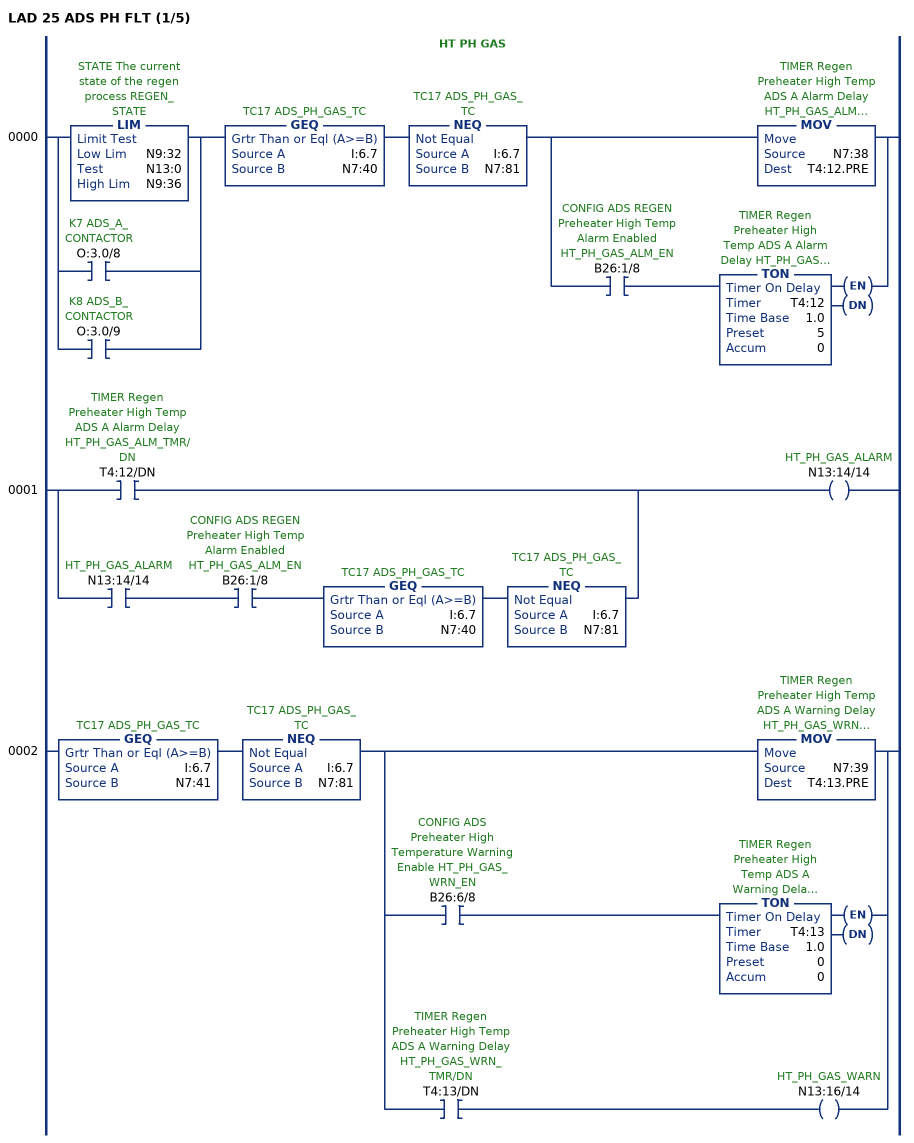
% Rung: 0 %
% TITLE: HT PH GAS %
SOR BST LIM N9:32 N13:0 N9:36 NXB XIC O:3.0/8 NXB XIC O:3.0/9 BND GEQ I:6.7 N7:40 NEQ I:6.7 N7:81 BST MOV N7:38 T4:12.PRE NXB XIC B26:1/8 TON T4:12 1.0 5 0 BND EOR
%   N9:32  REGEN_VENT  "STATE Regen Vent" %
%   N13:0  REGEN_STATE  "STATE The current state of the regen process" %
%   N9:36  REGEN_COOL  "STATE Regen Cool" %
%   O:3.0/8  ADS_A_CONTACTOR  "K7" %
%   O:3.0/9  ADS_B_CONTACTOR  "K8" %
%   I:6.7  ADS_PH_GAS_TC  "TC17" %
%   N7:40  HT_PH_GAS_ALM_SP  "CONFIG ADS Preheater High Temperature Alarm Temperature" %
%   N7:81  TC_OPEN_SP  "CONFIG The value read by an open TC input" %
%   N7:38  HT_PH_GAS_ALM_DLY  "CONFIG ADS Preheater High Temperature Alarm Delay" %
%   T4:12  HT_PH_GAS_ALM_TMR  "TIMER Regen Preheater High Temp ADS A Alarm Delay" %
%   B26:1/8  HT_PH_GAS_ALM_EN  "CONFIG ADS REGEN Preheater High Temp Alarm Enabled" %
% Rung: 1 %
SOR BST XIC T4:12/DN NXB XIC N13:14/14 XIC B26:1/8 GEQ I:6.7 N7:40 NEQ I:6.7 N7:81 BND OTE N13:14/14 EOR
%   T4:12  HT_PH_GAS_ALM_TMR  "TIMER Regen Preheater High Temp ADS A Alarm Delay" %
%   N13:14/14  HT_PH_GAS_ALARM %
%   B26:1/8  HT_PH_GAS_ALM_EN  "CONFIG ADS REGEN Preheater High Temp Alarm Enabled" %
%   I:6.7  ADS_PH_GAS_TC  "TC17" %
%   N7:40  HT_PH_GAS_ALM_SP  "CONFIG ADS Preheater High Temperature Alarm Temperature" %
%   N7:81  TC_OPEN_SP  "CONFIG The value read by an open TC input" %
% Rung: 2 %
SOR GEQ I:6.7 N7:41 NEQ I:6.7 N7:81 BST MOV N7:39 T4:13.PRE NXB XIC B26:6/8 TON T4:13 1.0 0 0 NXB XIC T4:13/DN OTE N13:16/14 BND EOR
%   I:6.7  ADS_PH_GAS_TC  "TC17" %
%   N7:41  HT_PH_GAS_WRN_SP  "CONFIG ADS Preheater High Temperature Warning Temperature" %
%   N7:81  TC_OPEN_SP  "CONFIG The value read by an open TC input" %
%   N7:39  HT_PH_GAS_WRN_DLY  "CONFIG ADS Preheater High Temperature Warning Delay" %
%   T4:13  HT_PH_GAS_WRN_TMR  "TIMER Regen Preheater High Temp ADS A Warning Delay" %
%   B26:6/8  HT_PH_GAS_WRN_EN  "CONFIG ADS Preheater High Temperature Warning Enable" %
%   N13:16/14  HT_PH_GAS_WARN %

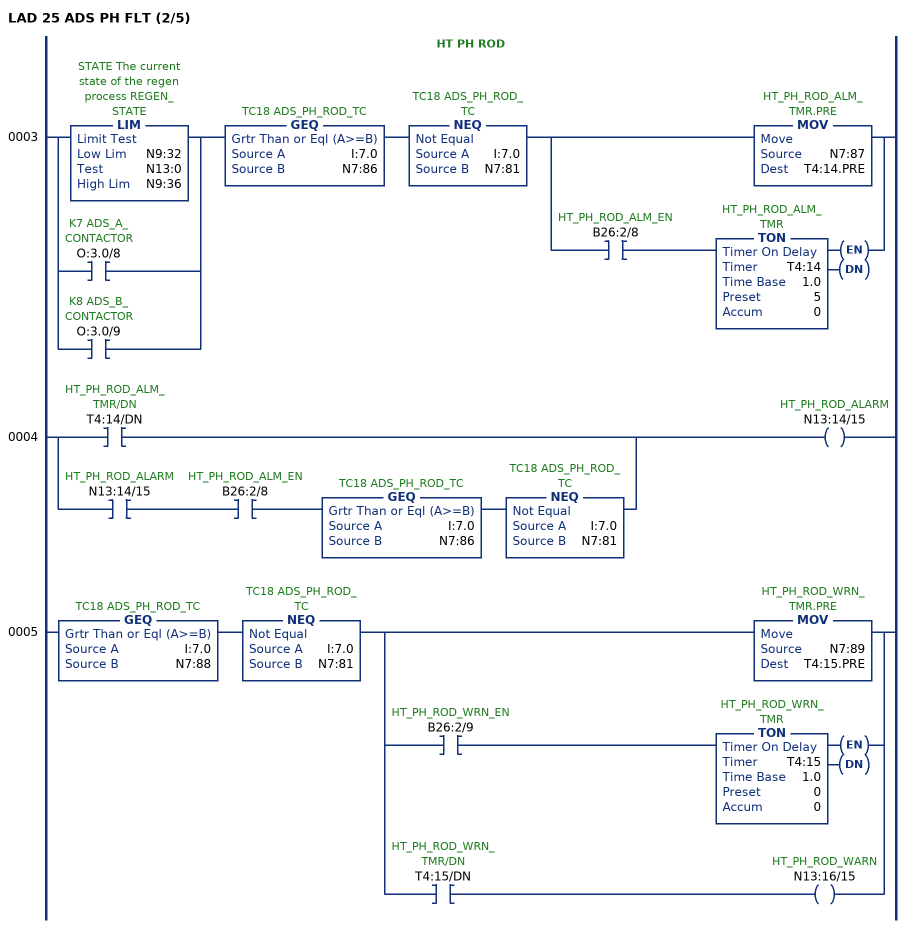
% Rung: 3 %
% TITLE: HT PH ROD %
SOR BST LIM N9:32 N13:0 N9:36 NXB XIC O:3.0/8 NXB XIC O:3.0/9 BND GEQ I:7.0 N7:86 NEQ I:7.0 N7:81 BST MOV N7:87 T4:14.PRE NXB XIC B26:2/8 TON T4:14 1.0 5 0 BND EOR
%   N9:32  REGEN_VENT  "STATE Regen Vent" %
%   N13:0  REGEN_STATE  "STATE The current state of the regen process" %
%   N9:36  REGEN_COOL  "STATE Regen Cool" %
%   O:3.0/8  ADS_A_CONTACTOR  "K7" %
%   O:3.0/9  ADS_B_CONTACTOR  "K8" %
%   I:7.0  ADS_PH_ROD_TC  "TC18" %
%   N7:86  HT_PH_ROD_ALM_SP %
%   N7:81  TC_OPEN_SP  "CONFIG The value read by an open TC input" %
%   N7:87  HT_PH_ROD_ALM_DLY %
%   T4:14  HT_PH_ROD_ALM_TMR %
%   B26:2/8  HT_PH_ROD_ALM_EN %
% Rung: 4 %
SOR BST XIC T4:14/DN NXB XIC N13:14/15 XIC B26:2/8 GEQ I:7.0 N7:86 NEQ I:7.0 N7:81 BND OTE N13:14/15 EOR
%   T4:14  HT_PH_ROD_ALM_TMR %
%   N13:14/15  HT_PH_ROD_ALARM %
%   B26:2/8  HT_PH_ROD_ALM_EN %
%   I:7.0  ADS_PH_ROD_TC  "TC18" %
%   N7:86  HT_PH_ROD_ALM_SP %
%   N7:81  TC_OPEN_SP  "CONFIG The value read by an open TC input" %
% Rung: 5 %
SOR GEQ I:7.0 N7:88 NEQ I:7.0 N7:81 BST MOV N7:89 T4:15.PRE NXB XIC B26:2/9 TON T4:15 1.0 0 0 NXB XIC T4:15/DN OTE N13:16/15 BND EOR
%   I:7.0  ADS_PH_ROD_TC  "TC18" %
%   N7:88  HT_PH_ROD_WRN_SP %
%   N7:81  TC_OPEN_SP  "CONFIG The value read by an open TC input" %
%   N7:89  HT_PH_ROD_WRN_DLY %
%   T4:15  HT_PH_ROD_WRN_TMR %
%   B26:2/9  HT_PH_ROD_WRN_EN %
%   N13:16/15  HT_PH_ROD_WARN %

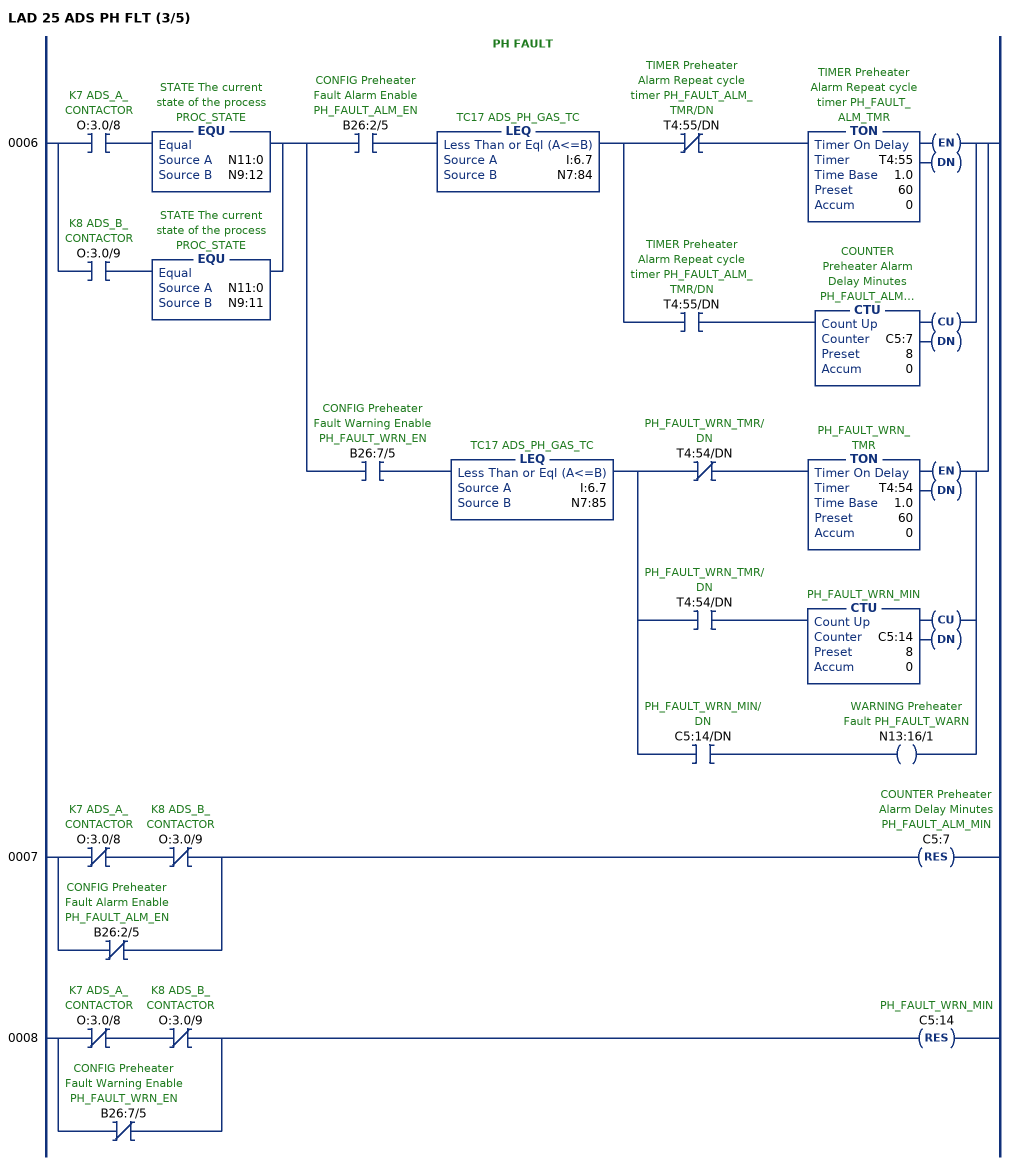
% Rung: 6 %
% TITLE: PH FAULT %
SOR BST XIC O:3.0/8 EQU N11:0 N9:12 NXB XIC O:3.0/9 EQU N11:0 N9:11 BND BST XIC B26:2/5 LEQ I:6.7 N7:84 BST XIO T4:55/DN TON T4:55 1.0 60 0 NXB XIC T4:55/DN CTU C5:7 8 0 BND NXB XIC B26:7/5 LEQ I:6.7 N7:85 BST XIO T4:54/DN TON T4:54 1.0 60 0 NXB XIC T4:54/DN CTU C5:14 8 0 NXB XIC C5:14/DN OTE N13:16/1 BND BND EOR
%   O:3.0/8  ADS_A_CONTACTOR  "K7" %
%   N11:0  PROC_STATE  "STATE The current state of the process" %
%   N9:12  PROC_PFY_B_REG_A  "STATE Process Purify B" %
%   O:3.0/9  ADS_B_CONTACTOR  "K8" %
%   N9:11  PROC_PFY_A_REG_B  "STATE Process Purify A" %
%   B26:2/5  PH_FAULT_ALM_EN  "CONFIG Preheater Fault Alarm Enable" %
%   I:6.7  ADS_PH_GAS_TC  "TC17" %
%   N7:84  PH_FAULT_ALARM_SP  "CONFIG Preheater Temperature Delta Alarm Setpoint" %
%   T4:55  PH_FAULT_ALM_TMR  "TIMER Preheater Alarm Repeat cycle timer" %
%   C5:7  PH_FAULT_ALM_MIN  "COUNTER Preheater Alarm Delay Minutes" %
%   B26:7/5  PH_FAULT_WRN_EN  "CONFIG Preheater Fault Warning Enable" %
%   N7:85  PH_FAULT_WARN_SP %
%   T4:54  PH_FAULT_WRN_TMR %
%   C5:14  PH_FAULT_WRN_MIN %
%   N13:16/1  PH_FAULT_WARN  "WARNING Preheater Fault" %
% Rung: 7 %
SOR BST XIO O:3.0/8 XIO O:3.0/9 NXB XIO B26:2/5 BND RES C5:7 EOR
%   O:3.0/8  ADS_A_CONTACTOR  "K7" %
%   O:3.0/9  ADS_B_CONTACTOR  "K8" %
%   B26:2/5  PH_FAULT_ALM_EN  "CONFIG Preheater Fault Alarm Enable" %
%   C5:7  PH_FAULT_ALM_MIN  "COUNTER Preheater Alarm Delay Minutes" %
% Rung: 8 %
SOR BST XIO O:3.0/8 XIO O:3.0/9 NXB XIO B26:7/5 BND RES C5:14 EOR
%   O:3.0/8  ADS_A_CONTACTOR  "K7" %
%   O:3.0/9  ADS_B_CONTACTOR  "K8" %
%   B26:7/5  PH_FAULT_WRN_EN  "CONFIG Preheater Fault Warning Enable" %
%   C5:14  PH_FAULT_WRN_MIN %

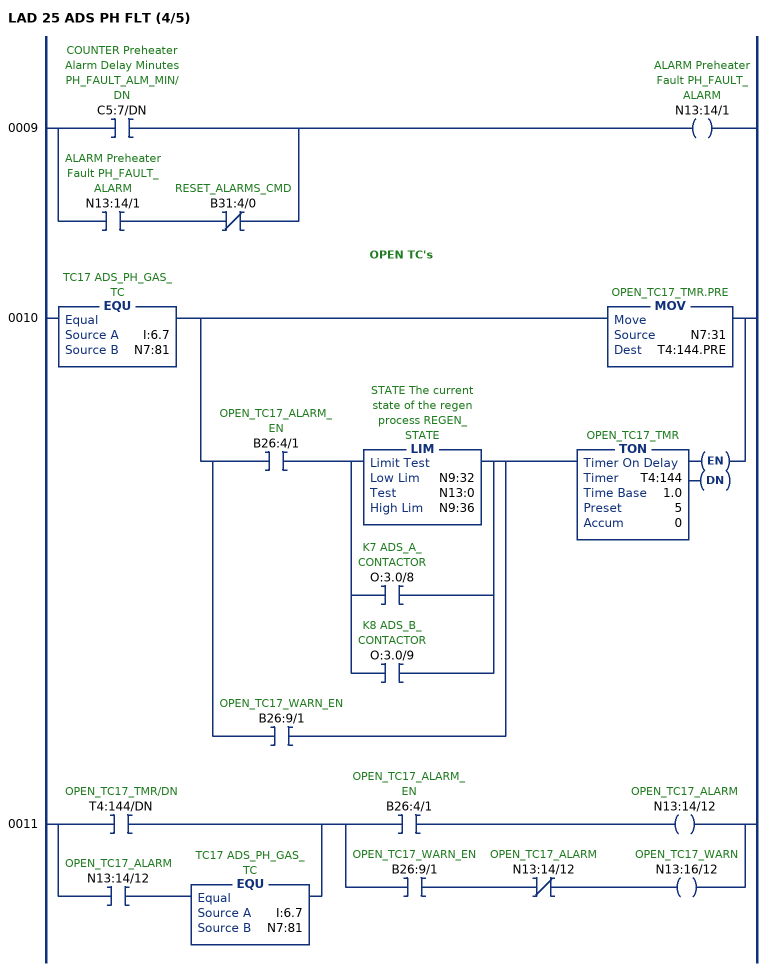
% Rung: 9 %
SOR BST XIC C5:7/DN NXB XIC N13:14/1 XIO B31:4/0 BND OTE N13:14/1 EOR
%   C5:7  PH_FAULT_ALM_MIN  "COUNTER Preheater Alarm Delay Minutes" %
%   N13:14/1  PH_FAULT_ALARM  "ALARM Preheater Fault" %
%   B31:4/0  RESET_ALARMS_CMD %
% Rung: 10 %
% TITLE: OPEN TC's %
SOR EQU I:6.7 N7:81 BST MOV N7:31 T4:144.PRE NXB BST XIC B26:4/1 BST LIM N9:32 N13:0 N9:36 NXB XIC O:3.0/8 NXB XIC O:3.0/9 BND NXB XIC B26:9/1 BND TON T4:144 1.0 5 0 BND EOR
%   I:6.7  ADS_PH_GAS_TC  "TC17" %
%   N7:81  TC_OPEN_SP  "CONFIG The value read by an open TC input" %
%   N7:31  OPEN_TC_DLY %
%   T4:144  OPEN_TC17_TMR %
%   B26:4/1  OPEN_TC17_ALARM_EN %
%   N9:32  REGEN_VENT  "STATE Regen Vent" %
%   N13:0  REGEN_STATE  "STATE The current state of the regen process" %
%   N9:36  REGEN_COOL  "STATE Regen Cool" %
%   O:3.0/8  ADS_A_CONTACTOR  "K7" %
%   O:3.0/9  ADS_B_CONTACTOR  "K8" %
%   B26:9/1  OPEN_TC17_WARN_EN %
% Rung: 11 %
SOR BST XIC T4:144/DN NXB XIC N13:14/12 EQU I:6.7 N7:81 BND BST XIC B26:4/1 OTE N13:14/12 NXB XIC B26:9/1 XIO N13:14/12 OTE N13:16/12 BND EOR
%   T4:144  OPEN_TC17_TMR %
%   N13:14/12  OPEN_TC17_ALARM %
%   I:6.7  ADS_PH_GAS_TC  "TC17" %
%   N7:81  TC_OPEN_SP  "CONFIG The value read by an open TC input" %
%   B26:4/1  OPEN_TC17_ALARM_EN %
%   B26:9/1  OPEN_TC17_WARN_EN %
%   N13:16/12  OPEN_TC17_WARN %

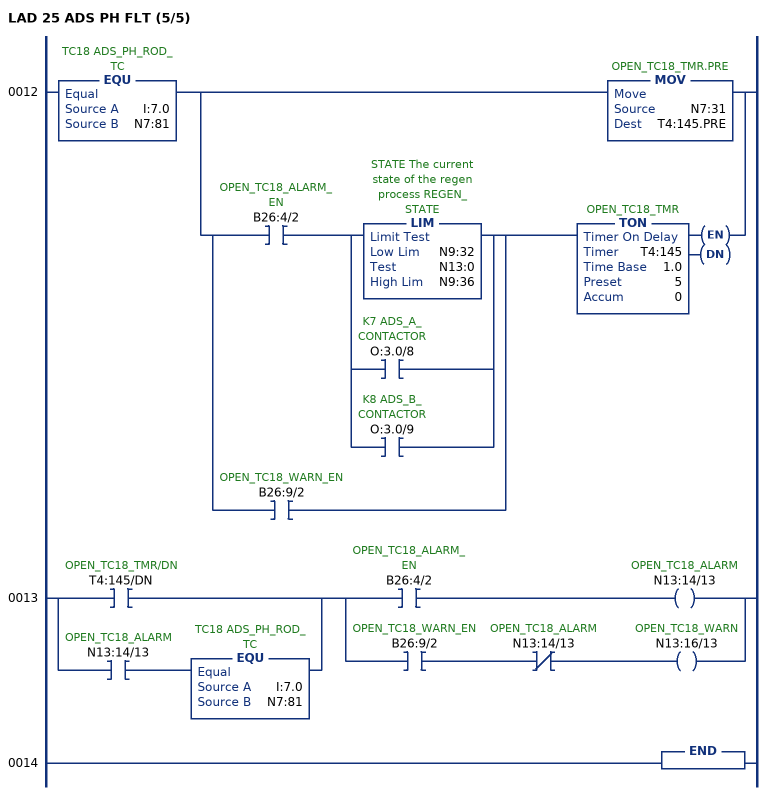
% Rung: 12 %
SOR EQU I:7.0 N7:81 BST MOV N7:31 T4:145.PRE NXB BST XIC B26:4/2 BST LIM N9:32 N13:0 N9:36 NXB XIC O:3.0/8 NXB XIC O:3.0/9 BND NXB XIC B26:9/2 BND TON T4:145 1.0 5 0 BND EOR
%   I:7.0  ADS_PH_ROD_TC  "TC18" %
%   N7:81  TC_OPEN_SP  "CONFIG The value read by an open TC input" %
%   N7:31  OPEN_TC_DLY %
%   T4:145  OPEN_TC18_TMR %
%   B26:4/2  OPEN_TC18_ALARM_EN %
%   N9:32  REGEN_VENT  "STATE Regen Vent" %
%   N13:0  REGEN_STATE  "STATE The current state of the regen process" %
%   N9:36  REGEN_COOL  "STATE Regen Cool" %
%   O:3.0/8  ADS_A_CONTACTOR  "K7" %
%   O:3.0/9  ADS_B_CONTACTOR  "K8" %
%   B26:9/2  OPEN_TC18_WARN_EN %
% Rung: 13 %
SOR BST XIC T4:145/DN NXB XIC N13:14/13 EQU I:7.0 N7:81 BND BST XIC B26:4/2 OTE N13:14/13 NXB XIC B26:9/2 XIO N13:14/13 OTE N13:16/13 BND EOR
%   T4:145  OPEN_TC18_TMR %
%   N13:14/13  OPEN_TC18_ALARM %
%   I:7.0  ADS_PH_ROD_TC  "TC18" %
%   N7:81  TC_OPEN_SP  "CONFIG The value read by an open TC input" %
%   B26:4/2  OPEN_TC18_ALARM_EN %
%   B26:9/2  OPEN_TC18_WARN_EN %
%   N13:16/13  OPEN_TC18_WARN %
% Rung: 14 %
SOR END EOR

LADDER 26 "GETTER"
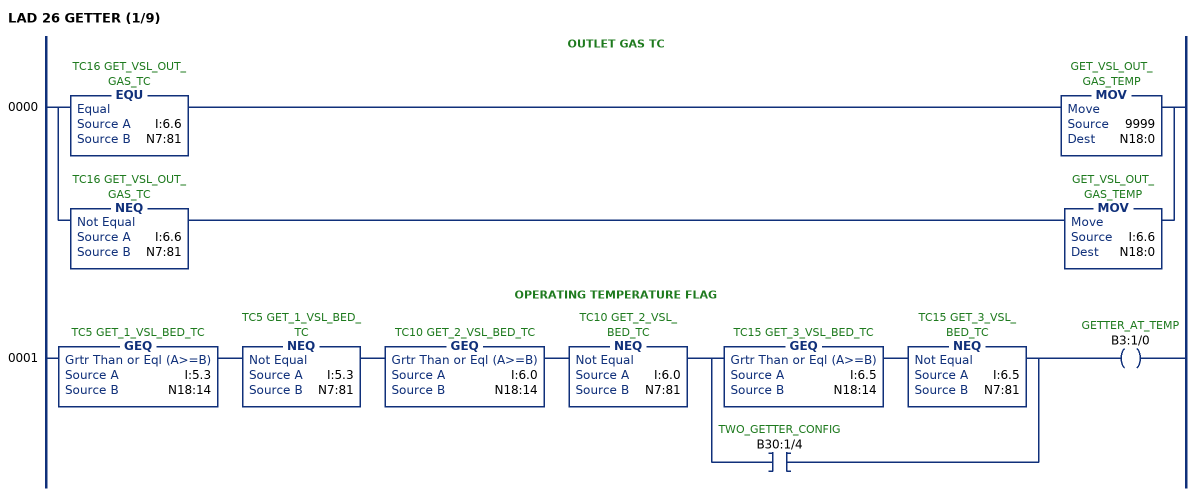
% Rung: 0 %
% TITLE: OUTLET GAS TC %
SOR BST EQU I:6.6 N7:81 MOV 9999 N18:0 NXB NEQ I:6.6 N7:81 MOV I:6.6 N18:0 BND EOR
%   I:6.6  GET_VSL_OUT_GAS_TC  "TC16" %
%   N7:81  TC_OPEN_SP  "CONFIG The value read by an open TC input" %
%   N18:0  GET_VSL_OUT_GAS_TEMP %
% Rung: 1 %
% TITLE: OPERATING TEMPERATURE FLAG %
SOR GEQ I:5.3 N18:14 NEQ I:5.3 N7:81 GEQ I:6.0 N18:14 NEQ I:6.0 N7:81 BST GEQ I:6.5 N18:14 NEQ I:6.5 N7:81 NXB XIC B30:1/4 BND OTE B3:1/0 EOR
%   I:5.3  GET_1_VSL_BED_TC  "TC5" %
%   N18:14  GETTER_OPERATING_TMP %
%   N7:81  TC_OPEN_SP  "CONFIG The value read by an open TC input" %
%   I:6.0  GET_2_VSL_BED_TC  "TC10" %
%   I:6.5  GET_3_VSL_BED_TC  "TC15" %
%   B30:1/4  TWO_GETTER_CONFIG %
%   B3:1/0  GETTER_AT_TEMP %

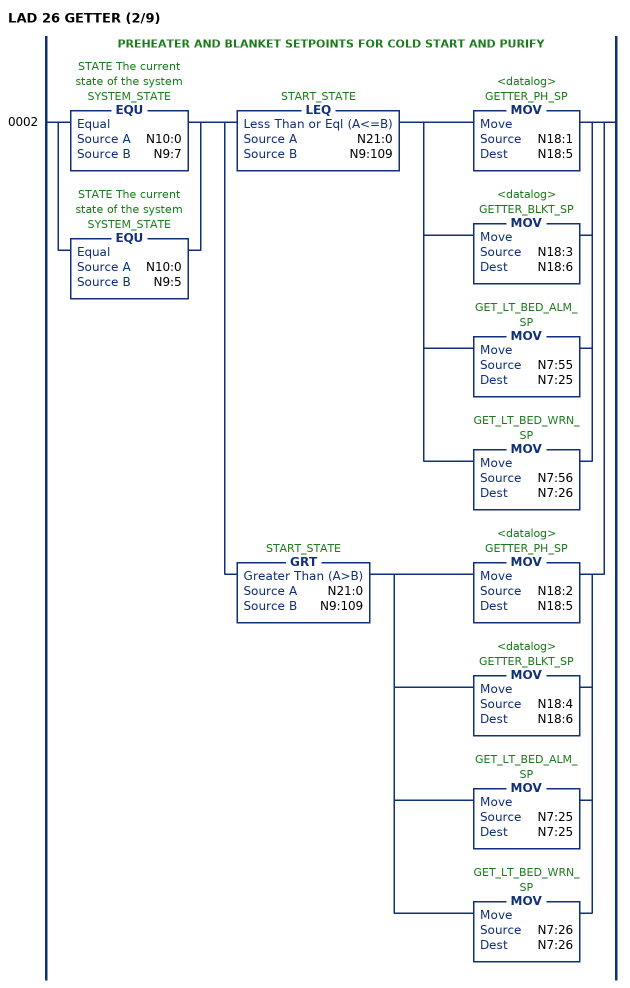
% Rung: 2 %
% TITLE: PREHEATER AND BLANKET SETPOINTS FOR COLD START AND PURIFY %
SOR BST EQU N10:0 N9:7 NXB EQU N10:0 N9:5 BND BST LEQ N21:0 N9:109 BST MOV N18:1 N18:5 NXB MOV N18:3 N18:6 NXB MOV N7:55 N7:25 NXB MOV N7:56 N7:26 BND NXB GRT N21:0 N9:109 BST MOV N18:2 N18:5 NXB MOV N18:4 N18:6 NXB MOV N7:25 N7:25 NXB MOV N7:26 N7:26 BND BND EOR
%   N10:0  SYSTEM_STATE  "STATE The current state of the system" %
%   N9:7  SYSTEM_COLD_START %
%   N9:5  SYSTEM_QUICK_START %
%   N21:0  START_STATE %
%   N9:109  START_BACKFILL_2 %
%   N18:1  GETTER_COLD_PH_SP %
%   N18:5  GETTER_PH_SP  "<datalog>" %
%   N18:3  GETTER_COLD_BLKT_SP %
%   N18:6  GETTER_BLKT_SP  "<datalog>" %
%   N7:55  GET_LT_BED_ST_ALM_SP %
%   N7:25  GET_LT_BED_ALM_SP %
%   N7:56  GET_LT_BED_ST_WRN_SP %
%   N7:26  GET_LT_BED_WRN_SP %
%   N18:2  GETTER_PFY_PH_SP %
%   N18:4  GETTER_PFY_BLKT_SP %

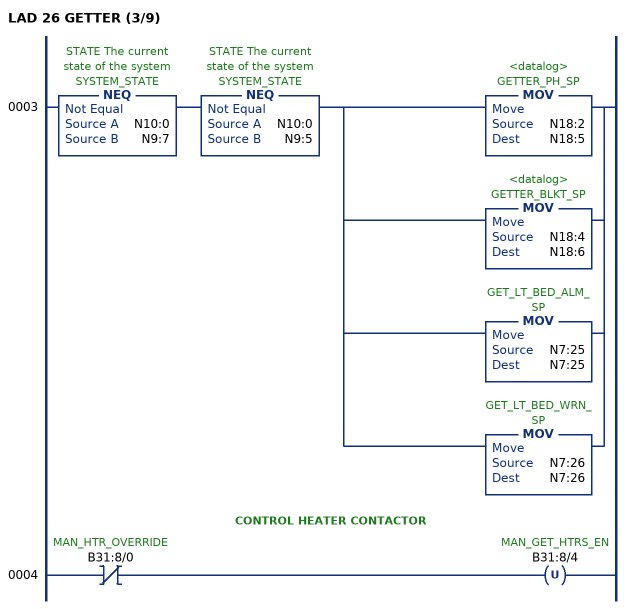
% Rung: 3 %
SOR NEQ N10:0 N9:7 NEQ N10:0 N9:5 BST MOV N18:2 N18:5 NXB MOV N18:4 N18:6 NXB MOV N7:25 N7:25 NXB MOV N7:26 N7:26 BND EOR
%   N10:0  SYSTEM_STATE  "STATE The current state of the system" %
%   N9:7  SYSTEM_COLD_START %
%   N9:5  SYSTEM_QUICK_START %
%   N18:2  GETTER_PFY_PH_SP %
%   N18:5  GETTER_PH_SP  "<datalog>" %
%   N18:4  GETTER_PFY_BLKT_SP %
%   N18:6  GETTER_BLKT_SP  "<datalog>" %
%   N7:25  GET_LT_BED_ALM_SP %
%   N7:26  GET_LT_BED_WRN_SP %
% Rung: 4 %
% TITLE: CONTROL HEATER CONTACTOR %
SOR XIO B31:8/0 OTU B31:8/4 EOR
%   B31:8/0  MAN_HTR_OVERRIDE %
%   B31:8/4  MAN_GET_HTRS_EN %

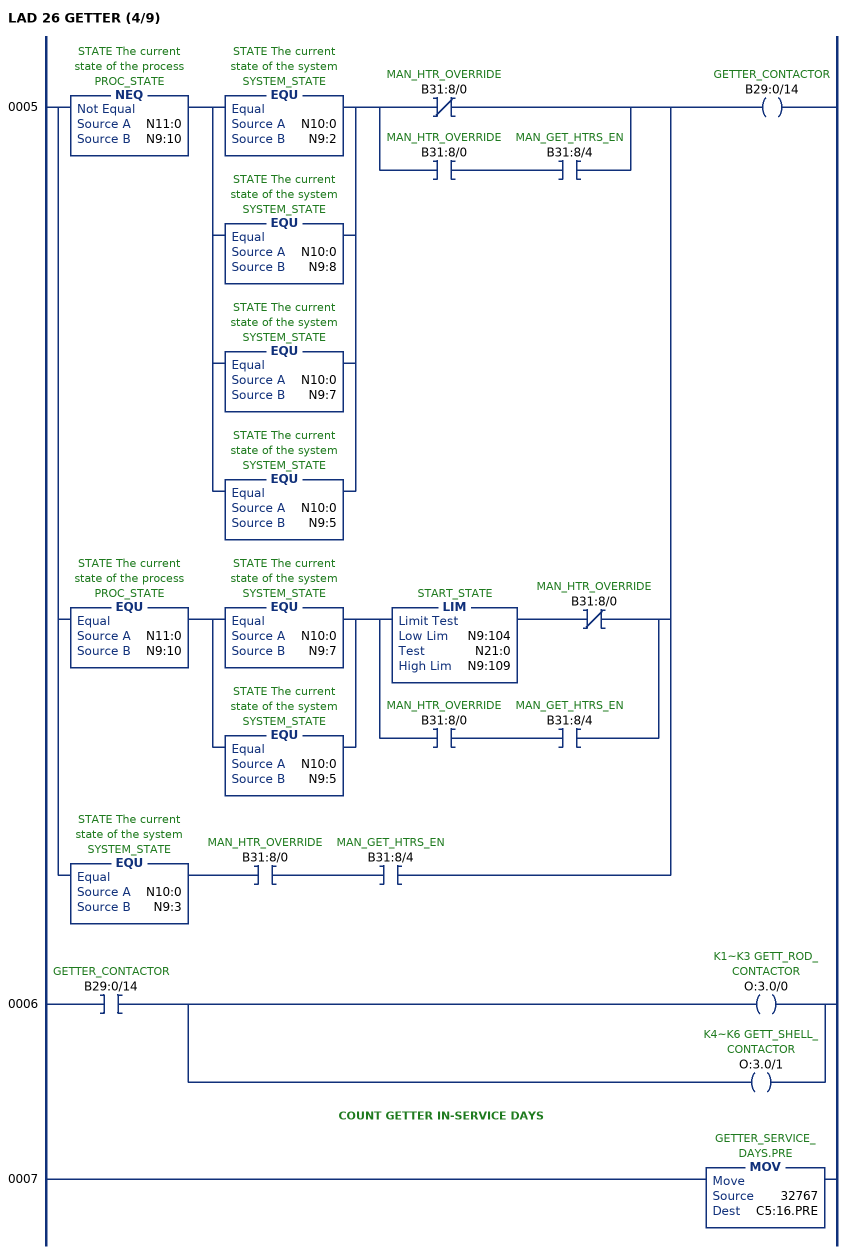
% Rung: 5 %
SOR BST NEQ N11:0 N9:10 BST EQU N10:0 N9:2 NXB EQU N10:0 N9:8 NXB EQU N10:0 N9:7 NXB EQU N10:0 N9:5 BND BST XIO B31:8/0 NXB XIC B31:8/0 XIC B31:8/4 BND NXB EQU N11:0 N9:10 BST EQU N10:0 N9:7 NXB EQU N10:0 N9:5 BND BST LIM N9:104 N21:0 N9:109 XIO B31:8/0 NXB XIC B31:8/0 XIC B31:8/4 BND NXB EQU N10:0 N9:3 XIC B31:8/0 XIC B31:8/4 BND OTE B29:0/14 EOR
%   N11:0  PROC_STATE  "STATE The current state of the process" %
%   N9:10  PROC_STANDBY  "STATE Process Standby" %
%   N10:0  SYSTEM_STATE  "STATE The current state of the system" %
%   N9:2  SYSTEM_PROCESS  "STATE System Process" %
%   N9:8  SYSTEM_SUPPLEMENTAL %
%   N9:7  SYSTEM_COLD_START %
%   N9:5  SYSTEM_QUICK_START %
%   B31:8/0  MAN_HTR_OVERRIDE %
%   B31:8/4  MAN_GET_HTRS_EN %
%   N9:104  START_HEAT %
%   N21:0  START_STATE %
%   N9:109  START_BACKFILL_2 %
%   N9:3  SYSTEM_MANUAL  "STATE System Manual" %
%   B29:0/14  GETTER_CONTACTOR %
% Rung: 6 %
SOR XIC B29:0/14 BST OTE O:3.0/0 NXB OTE O:3.0/1 BND EOR
%   B29:0/14  GETTER_CONTACTOR %
%   O:3.0/0  GETT_ROD_CONTACTOR  "K1~K3" %
%   O:3.0/1  GETT_SHELL_CONTACTOR  "K4~K6" %
% Rung: 7 %
% TITLE: COUNT GETTER IN-SERVICE DAYS %
SOR MOV 32767 C5:16.PRE EOR
%   C5:16  GETTER_SERVICE_DAYS %

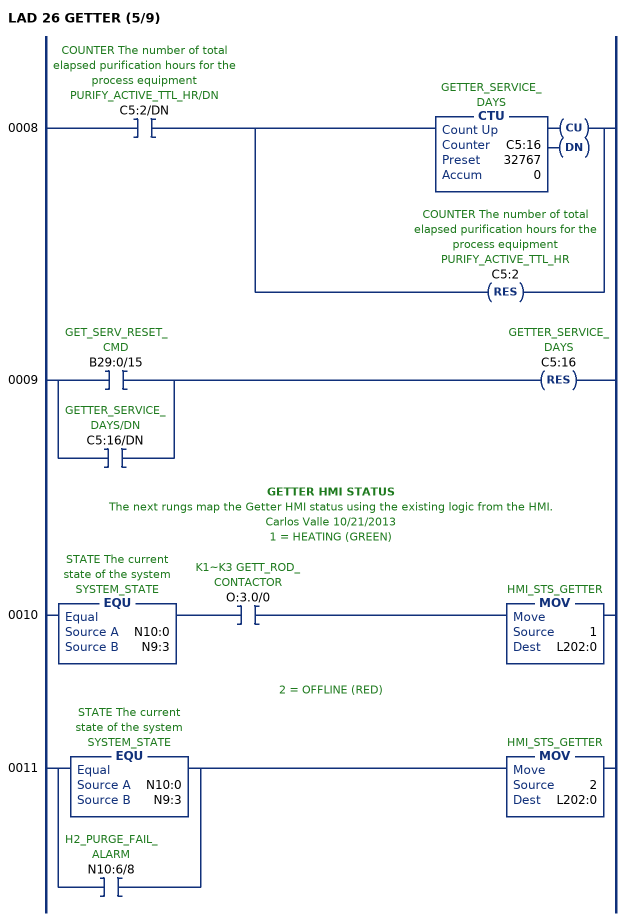
% Rung: 8 %
SOR XIC C5:2/DN BST CTU C5:16 32767 0 NXB RES C5:2 BND EOR
%   C5:2  PURIFY_ACTIVE_TTL_HR  "COUNTER The number of total elapsed purification hours for the process equipment" %
%   C5:16  GETTER_SERVICE_DAYS %
% Rung: 9 %
SOR BST XIC B29:0/15 NXB XIC C5:16/DN BND RES C5:16 EOR
%   B29:0/15  GET_SERV_RESET_CMD %
%   C5:16  GETTER_SERVICE_DAYS %
% Rung: 10 %
% TITLE: GETTER HMI STATUS %
% The next rungs map the Getter HMI status using the existing logic from the HMI.
% Carlos Valle 10/21/2013
% 1 = HEATING (GREEN) %
SOR EQU N10:0 N9:3 XIC O:3.0/0 MOV 1 L202:0 EOR
%   N10:0  SYSTEM_STATE  "STATE The current state of the system" %
%   N9:3  SYSTEM_MANUAL  "STATE System Manual" %
%   O:3.0/0  GETT_ROD_CONTACTOR  "K1~K3" %
%   L202:0  HMI_STS_GETTER %
% Rung: 11 %
% 2 = OFFLINE (RED) %
SOR BST EQU N10:0 N9:3 NXB XIC N10:6/8 BND MOV 2 L202:0 EOR
%   N10:0  SYSTEM_STATE  "STATE The current state of the system" %
%   N9:3  SYSTEM_MANUAL  "STATE System Manual" %
%   N10:6/8  H2_PURGE_FAIL_ALARM %
%   L202:0  HMI_STS_GETTER %

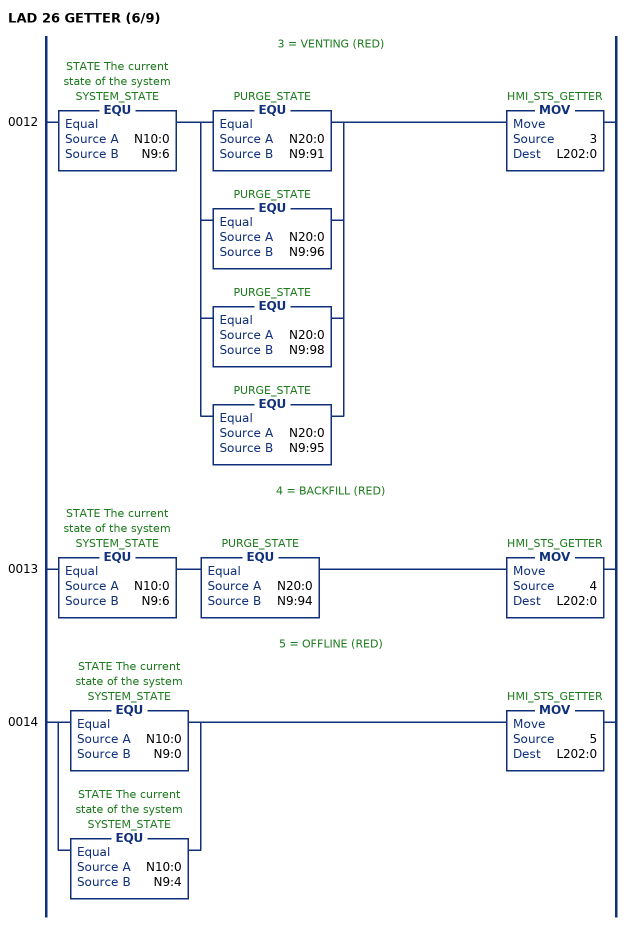
% Rung: 12 %
% 3 = VENTING (RED) %
SOR EQU N10:0 N9:6 BST EQU N20:0 N9:91 NXB EQU N20:0 N9:96 NXB EQU N20:0 N9:98 NXB EQU N20:0 N9:95 BND MOV 3 L202:0 EOR
%   N10:0  SYSTEM_STATE  "STATE The current state of the system" %
%   N9:6  SYSTEM_PURGE %
%   N20:0  PURGE_STATE %
%   N9:91  PURGE_INIT_VENT %
%   N9:96  PURGE_DONE %
%   N9:98  PURGE_VENT_GET_2 %
%   N9:95  PURGE_FINAL_VENT %
%   L202:0  HMI_STS_GETTER %
% Rung: 13 %
% 4 = BACKFILL (RED) %
SOR EQU N10:0 N9:6 EQU N20:0 N9:94 MOV 4 L202:0 EOR
%   N10:0  SYSTEM_STATE  "STATE The current state of the system" %
%   N9:6  SYSTEM_PURGE %
%   N20:0  PURGE_STATE %
%   N9:94  PURGE_BACKFILL %
%   L202:0  HMI_STS_GETTER %
% Rung: 14 %
% 5 = OFFLINE (RED) %
SOR BST EQU N10:0 N9:0 NXB EQU N10:0 N9:4 BND MOV 5 L202:0 EOR
%   N10:0  SYSTEM_STATE  "STATE The current state of the system" %
%   N9:0  SYSTEM_OFFLINE %
%   N9:4  SYSTEM_ALARM  "STATE System Alarm" %
%   L202:0  HMI_STS_GETTER %

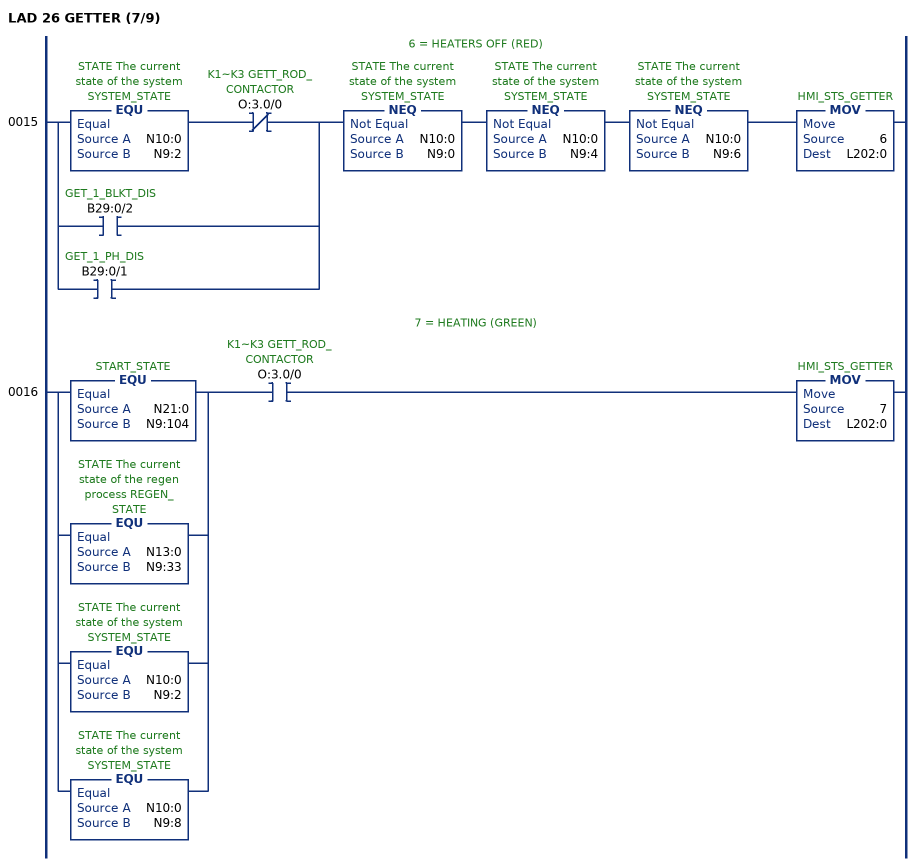
% Rung: 15 %
% 6 = HEATERS OFF (RED) %
SOR BST EQU N10:0 N9:2 XIO O:3.0/0 NXB XIC B29:0/2 NXB XIC B29:0/1 BND NEQ N10:0 N9:0 NEQ N10:0 N9:4 NEQ N10:0 N9:6 MOV 6 L202:0 EOR
%   N10:0  SYSTEM_STATE  "STATE The current state of the system" %
%   N9:2  SYSTEM_PROCESS  "STATE System Process" %
%   O:3.0/0  GETT_ROD_CONTACTOR  "K1~K3" %
%   B29:0/2  GET_1_BLKT_DIS %
%   B29:0/1  GET_1_PH_DIS %
%   N9:0  SYSTEM_OFFLINE %
%   N9:4  SYSTEM_ALARM  "STATE System Alarm" %
%   N9:6  SYSTEM_PURGE %
%   L202:0  HMI_STS_GETTER %
% Rung: 16 %
% 7 = HEATING (GREEN) %
SOR BST EQU N21:0 N9:104 NXB EQU N13:0 N9:33 NXB EQU N10:0 N9:2 NXB EQU N10:0 N9:8 BND XIC O:3.0/0 MOV 7 L202:0 EOR
%   N21:0  START_STATE %
%   N9:104  START_HEAT %
%   N13:0  REGEN_STATE  "STATE The current state of the regen process" %
%   N9:33  REGEN_HEAT_BED  "STATE Regen Heat wall" %
%   N10:0  SYSTEM_STATE  "STATE The current state of the system" %
%   N9:2  SYSTEM_PROCESS  "STATE System Process" %
%   N9:8  SYSTEM_SUPPLEMENTAL %
%   O:3.0/0  GETT_ROD_CONTACTOR  "K1~K3" %
%   L202:0  HMI_STS_GETTER %

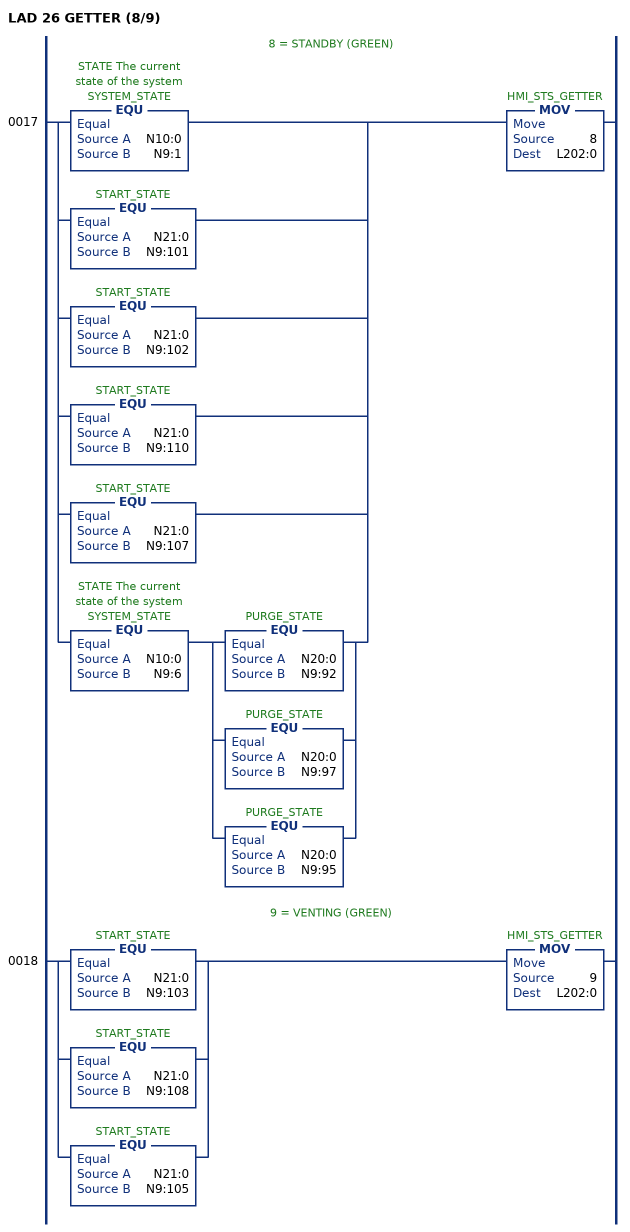
% Rung: 17 %
% 8 = STANDBY (GREEN) %
SOR BST EQU N10:0 N9:1 NXB EQU N21:0 N9:101 NXB EQU N21:0 N9:102 NXB EQU N21:0 N9:110 NXB EQU N21:0 N9:107 NXB EQU N10:0 N9:6 BST EQU N20:0 N9:92 NXB EQU N20:0 N9:97 NXB EQU N20:0 N9:95 BND BND MOV 8 L202:0 EOR
%   N10:0  SYSTEM_STATE  "STATE The current state of the system" %
%   N9:1  SYSTEM_STANDBY  "STATE System Process" %
%   N21:0  START_STATE %
%   N9:101  START_COOL %
%   N9:102  START_VENT_ADS_1 %
%   N9:110  START_REG_VENT %
%   N9:107  START_VENT_ADS_2 %
%   N9:6  SYSTEM_PURGE %
%   N20:0  PURGE_STATE %
%   N9:92  PURGE_VENT_ADSORBER %
%   N9:97  PURGE_VENT_ADS_2 %
%   N9:95  PURGE_FINAL_VENT %
%   L202:0  HMI_STS_GETTER %
% Rung: 18 %
% 9 = VENTING (GREEN) %
SOR BST EQU N21:0 N9:103 NXB EQU N21:0 N9:108 NXB EQU N21:0 N9:105 BND MOV 9 L202:0 EOR
%   N21:0  START_STATE %
%   N9:103  START_VENT_GET_1 %
%   N9:108  START_VENT_GET_2 %
%   N9:105  START_VENT_ALL %
%   L202:0  HMI_STS_GETTER %

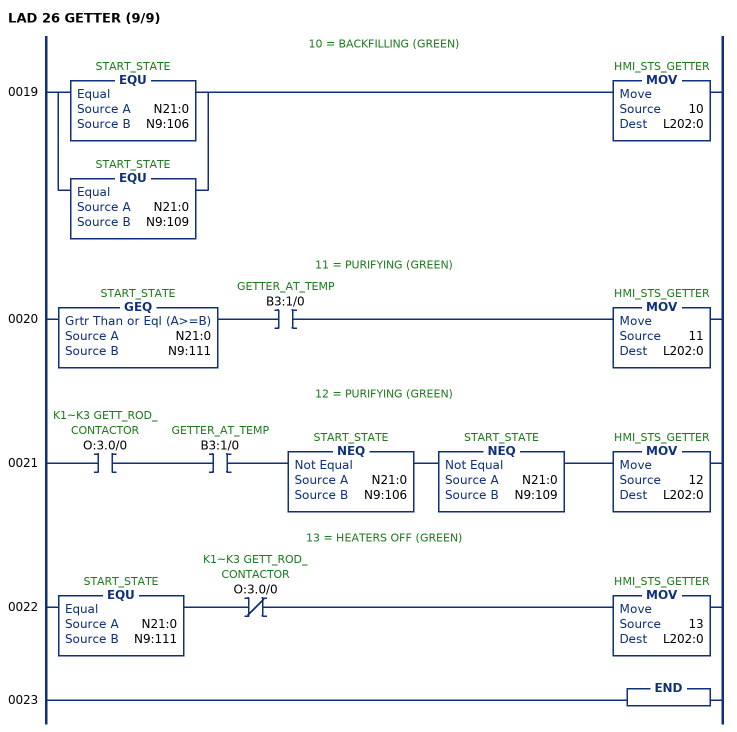
% Rung: 19 %
% 10 = BACKFILLING (GREEN) %
SOR BST EQU N21:0 N9:106 NXB EQU N21:0 N9:109 BND MOV 10 L202:0 EOR
%   N21:0  START_STATE %
%   N9:106  START_BACKFILL_1 %
%   N9:109  START_BACKFILL_2 %
%   L202:0  HMI_STS_GETTER %
% Rung: 20 %
% 11 = PURIFYING (GREEN) %
SOR GEQ N21:0 N9:111 XIC B3:1/0 MOV 11 L202:0 EOR
%   N21:0  START_STATE %
%   N9:111  START_REG_HEAT %
%   B3:1/0  GETTER_AT_TEMP %
%   L202:0  HMI_STS_GETTER %
% Rung: 21 %
% 12 = PURIFYING (GREEN) %
SOR XIC O:3.0/0 XIC B3:1/0 NEQ N21:0 N9:106 NEQ N21:0 N9:109 MOV 12 L202:0 EOR
%   O:3.0/0  GETT_ROD_CONTACTOR  "K1~K3" %
%   B3:1/0  GETTER_AT_TEMP %
%   N21:0  START_STATE %
%   N9:106  START_BACKFILL_1 %
%   N9:109  START_BACKFILL_2 %
%   L202:0  HMI_STS_GETTER %
% Rung: 22 %
% 13 = HEATERS OFF (GREEN) %
SOR EQU N21:0 N9:111 XIO O:3.0/0 MOV 13 L202:0 EOR
%   N21:0  START_STATE %
%   N9:111  START_REG_HEAT %
%   O:3.0/0  GETT_ROD_CONTACTOR  "K1~K3" %
%   L202:0  HMI_STS_GETTER %
% Rung: 23 %
SOR END EOR

LADDER 27 "GET 1 FLT"
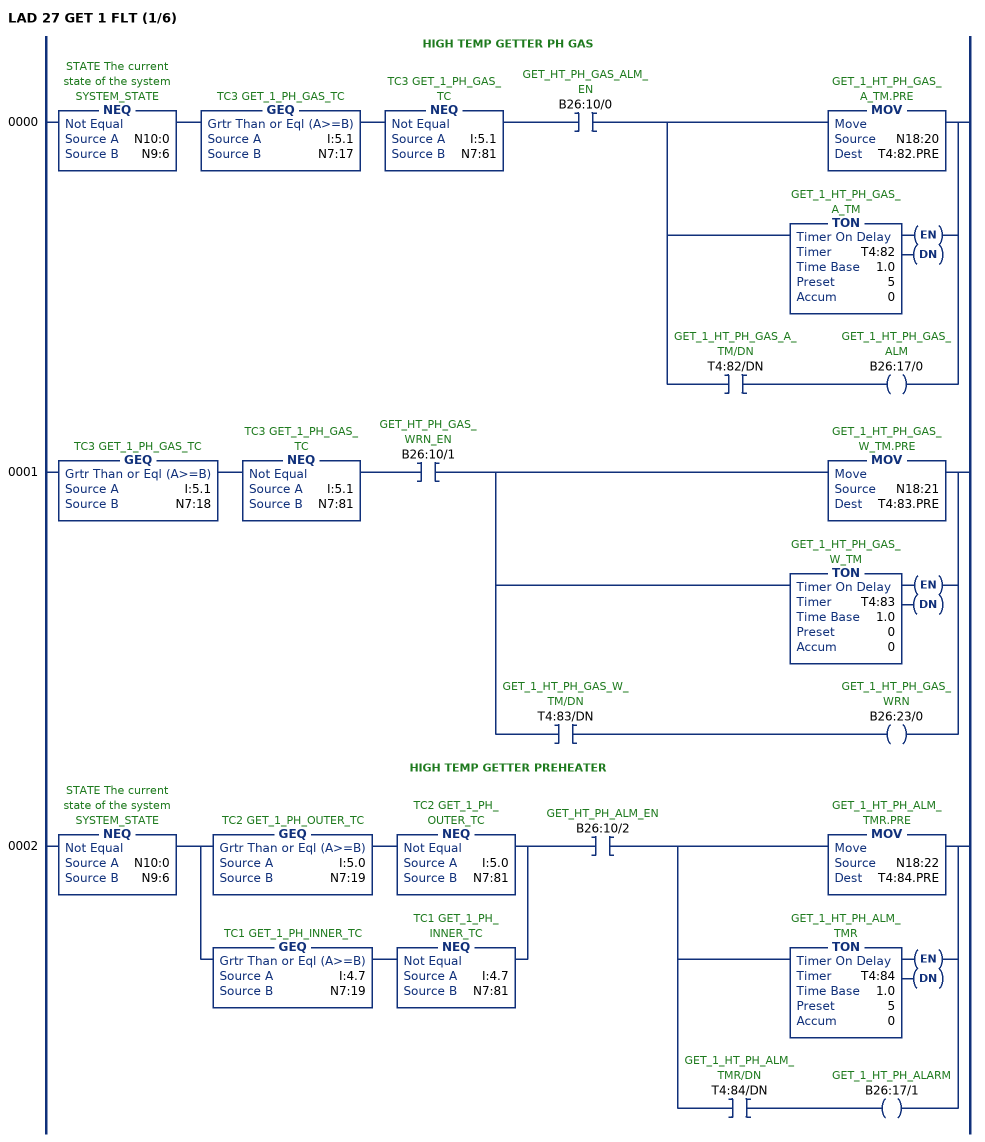
% Rung: 0 %
% TITLE: HIGH TEMP GETTER PH GAS %
SOR NEQ N10:0 N9:6 GEQ I:5.1 N7:17 NEQ I:5.1 N7:81 XIC B26:10/0 BST MOV N18:20 T4:82.PRE NXB TON T4:82 1.0 5 0 NXB XIC T4:82/DN OTE B26:17/0 BND EOR
%   N10:0  SYSTEM_STATE  "STATE The current state of the system" %
%   N9:6  SYSTEM_PURGE %
%   I:5.1  GET_1_PH_GAS_TC  "TC3" %
%   N7:17  GET_HT_PH_GAS_ALM_SP %
%   N7:81  TC_OPEN_SP  "CONFIG The value read by an open TC input" %
%   B26:10/0  GET_HT_PH_GAS_ALM_EN %
%   N18:20  GET_HT_PH_GAS_ALM_DL %
%   T4:82  GET_1_HT_PH_GAS_A_TM %
%   B26:17/0  GET_1_HT_PH_GAS_ALM %
% Rung: 1 %
SOR GEQ I:5.1 N7:18 NEQ I:5.1 N7:81 XIC B26:10/1 BST MOV N18:21 T4:83.PRE NXB TON T4:83 1.0 0 0 NXB XIC T4:83/DN OTE B26:23/0 BND EOR
%   I:5.1  GET_1_PH_GAS_TC  "TC3" %
%   N7:18  GET_HT_PH_GAS_WRN_SP %
%   N7:81  TC_OPEN_SP  "CONFIG The value read by an open TC input" %
%   B26:10/1  GET_HT_PH_GAS_WRN_EN %
%   N18:21  GET_HT_PH_GAS_WRN_DL %
%   T4:83  GET_1_HT_PH_GAS_W_TM %
%   B26:23/0  GET_1_HT_PH_GAS_WRN %
% Rung: 2 %
% TITLE: HIGH TEMP GETTER PREHEATER %
SOR NEQ N10:0 N9:6 BST GEQ I:5.0 N7:19 NEQ I:5.0 N7:81 NXB GEQ I:4.7 N7:19 NEQ I:4.7 N7:81 BND XIC B26:10/2 BST MOV N18:22 T4:84.PRE NXB TON T4:84 1.0 5 0 NXB XIC T4:84/DN OTE B26:17/1 BND EOR
%   N10:0  SYSTEM_STATE  "STATE The current state of the system" %
%   N9:6  SYSTEM_PURGE %
%   I:5.0  GET_1_PH_OUTER_TC  "TC2" %
%   N7:19  GET_HT_PH_ALM_SP %
%   N7:81  TC_OPEN_SP  "CONFIG The value read by an open TC input" %
%   I:4.7  GET_1_PH_INNER_TC  "TC1" %
%   B26:10/2  GET_HT_PH_ALM_EN %
%   N18:22  GET_HT_PH_ALM_DLY %
%   T4:84  GET_1_HT_PH_ALM_TMR %
%   B26:17/1  GET_1_HT_PH_ALARM %

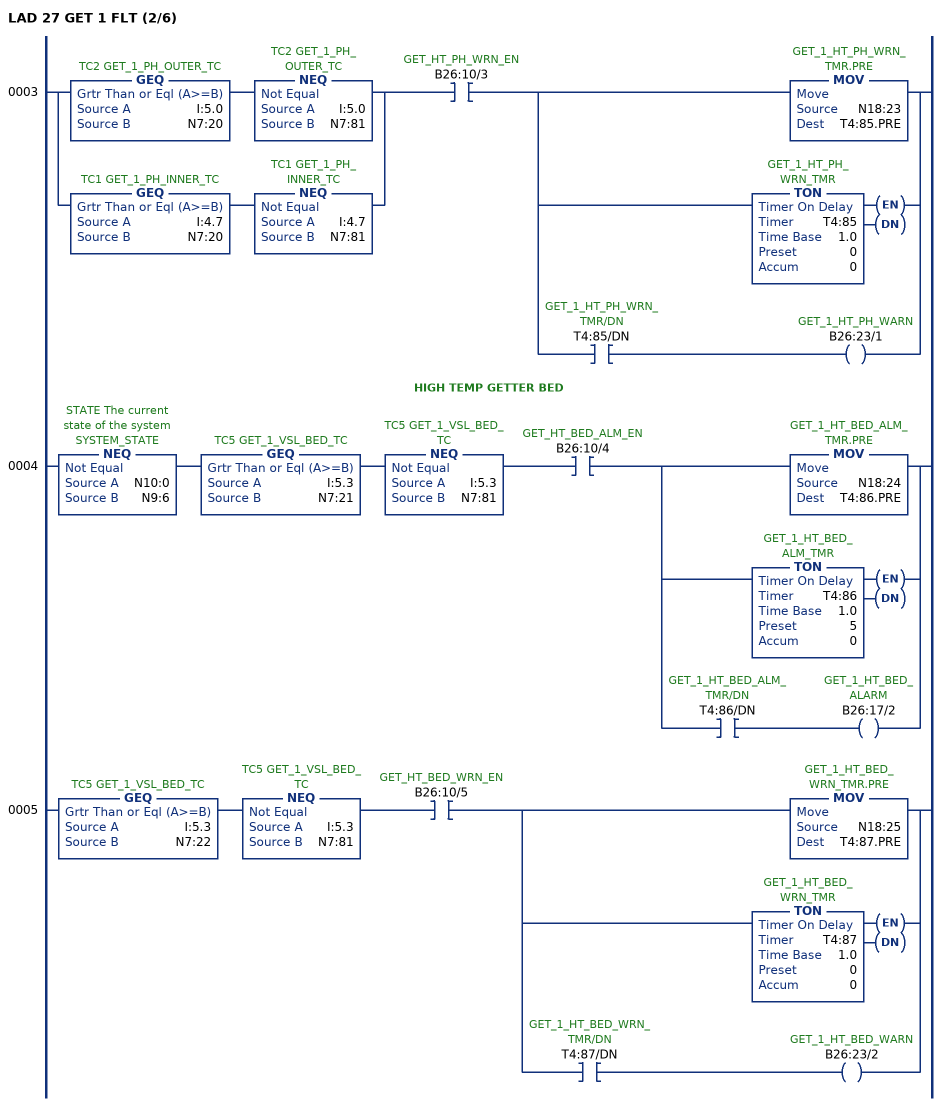
% Rung: 3 %
SOR BST GEQ I:5.0 N7:20 NEQ I:5.0 N7:81 NXB GEQ I:4.7 N7:20 NEQ I:4.7 N7:81 BND XIC B26:10/3 BST MOV N18:23 T4:85.PRE NXB TON T4:85 1.0 0 0 NXB XIC T4:85/DN OTE B26:23/1 BND EOR
%   I:5.0  GET_1_PH_OUTER_TC  "TC2" %
%   N7:20  GET_HT_PH_WRN_SP %
%   N7:81  TC_OPEN_SP  "CONFIG The value read by an open TC input" %
%   I:4.7  GET_1_PH_INNER_TC  "TC1" %
%   B26:10/3  GET_HT_PH_WRN_EN %
%   N18:23  GET_HT_PH_WRN_DLY %
%   T4:85  GET_1_HT_PH_WRN_TMR %
%   B26:23/1  GET_1_HT_PH_WARN %
% Rung: 4 %
% TITLE: HIGH TEMP GETTER BED %
SOR NEQ N10:0 N9:6 GEQ I:5.3 N7:21 NEQ I:5.3 N7:81 XIC B26:10/4 BST MOV N18:24 T4:86.PRE NXB TON T4:86 1.0 5 0 NXB XIC T4:86/DN OTE B26:17/2 BND EOR
%   N10:0  SYSTEM_STATE  "STATE The current state of the system" %
%   N9:6  SYSTEM_PURGE %
%   I:5.3  GET_1_VSL_BED_TC  "TC5" %
%   N7:21  GET_HT_BED_ALM_SP %
%   N7:81  TC_OPEN_SP  "CONFIG The value read by an open TC input" %
%   B26:10/4  GET_HT_BED_ALM_EN %
%   N18:24  GET_HT_BED_ALM_DLY %
%   T4:86  GET_1_HT_BED_ALM_TMR %
%   B26:17/2  GET_1_HT_BED_ALARM %
% Rung: 5 %
SOR GEQ I:5.3 N7:22 NEQ I:5.3 N7:81 XIC B26:10/5 BST MOV N18:25 T4:87.PRE NXB TON T4:87 1.0 0 0 NXB XIC T4:87/DN OTE B26:23/2 BND EOR
%   I:5.3  GET_1_VSL_BED_TC  "TC5" %
%   N7:22  GET_HT_BED_WRN_SP %
%   N7:81  TC_OPEN_SP  "CONFIG The value read by an open TC input" %
%   B26:10/5  GET_HT_BED_WRN_EN %
%   N18:25  GET_HT_BED_WRN_DLY %
%   T4:87  GET_1_HT_BED_WRN_TMR %
%   B26:23/2  GET_1_HT_BED_WARN %

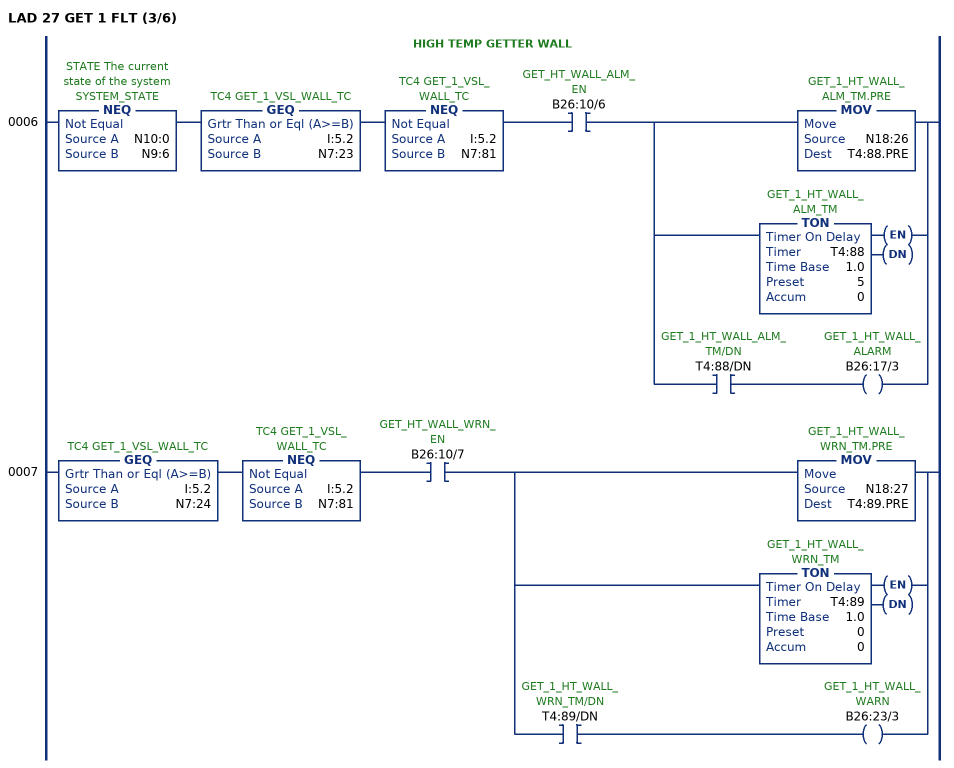
% Rung: 6 %
% TITLE: HIGH TEMP GETTER WALL %
SOR NEQ N10:0 N9:6 GEQ I:5.2 N7:23 NEQ I:5.2 N7:81 XIC B26:10/6 BST MOV N18:26 T4:88.PRE NXB TON T4:88 1.0 5 0 NXB XIC T4:88/DN OTE B26:17/3 BND EOR
%   N10:0  SYSTEM_STATE  "STATE The current state of the system" %
%   N9:6  SYSTEM_PURGE %
%   I:5.2  GET_1_VSL_WALL_TC  "TC4" %
%   N7:23  GET_HT_WALL_ALM_SP %
%   N7:81  TC_OPEN_SP  "CONFIG The value read by an open TC input" %
%   B26:10/6  GET_HT_WALL_ALM_EN %
%   N18:26  GET_HT_WALL_ALM_DLY %
%   T4:88  GET_1_HT_WALL_ALM_TM %
%   B26:17/3  GET_1_HT_WALL_ALARM %
% Rung: 7 %
SOR GEQ I:5.2 N7:24 NEQ I:5.2 N7:81 XIC B26:10/7 BST MOV N18:27 T4:89.PRE NXB TON T4:89 1.0 0 0 NXB XIC T4:89/DN OTE B26:23/3 BND EOR
%   I:5.2  GET_1_VSL_WALL_TC  "TC4" %
%   N7:24  GET_HT_WALL_WRN_SP %
%   N7:81  TC_OPEN_SP  "CONFIG The value read by an open TC input" %
%   B26:10/7  GET_HT_WALL_WRN_EN %
%   N18:27  GET_HT_WALL_WRN_DLY %
%   T4:89  GET_1_HT_WALL_WRN_TM %
%   B26:23/3  GET_1_HT_WALL_WARN %

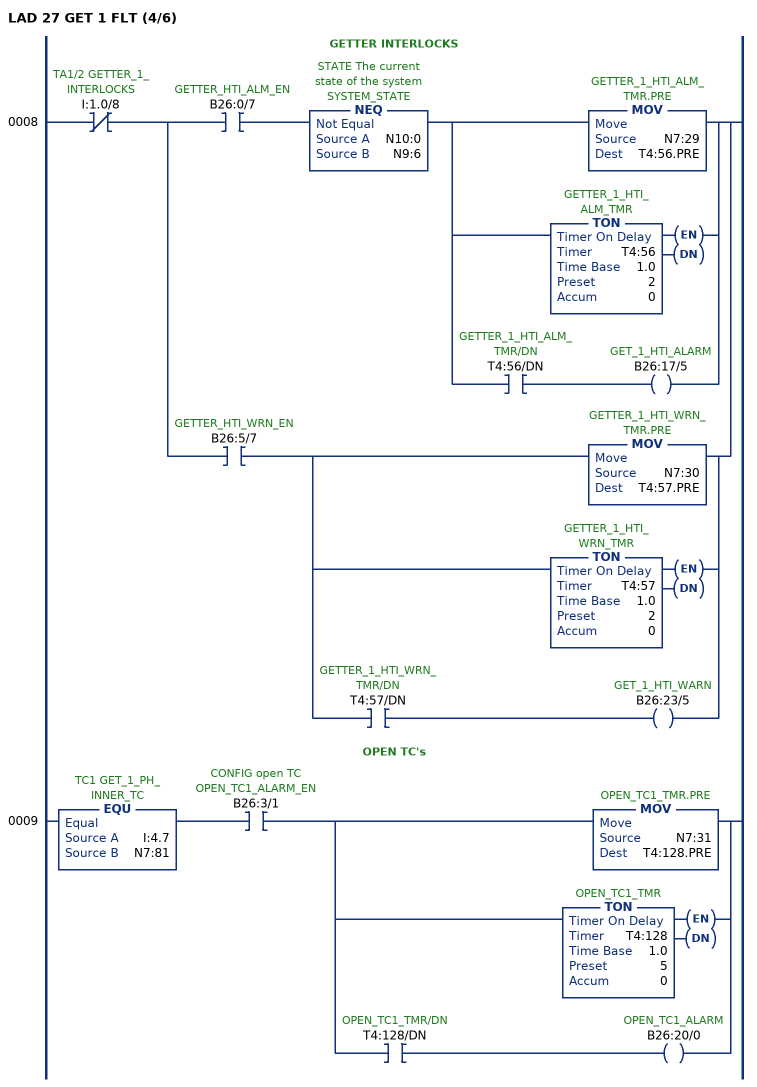
% Rung: 8 %
% TITLE: GETTER INTERLOCKS %
SOR XIO I:1.0/8 BST XIC B26:0/7 NEQ N10:0 N9:6 BST MOV N7:29 T4:56.PRE NXB TON T4:56 1.0 2 0 NXB XIC T4:56/DN OTE B26:17/5 BND NXB XIC B26:5/7 BST MOV N7:30 T4:57.PRE NXB TON T4:57 1.0 2 0 NXB XIC T4:57/DN OTE B26:23/5 BND BND EOR
%   I:1.0/8  GETTER_1_INTERLOCKS  "TA1/2" %
%   B26:0/7  GETTER_HTI_ALM_EN %
%   N10:0  SYSTEM_STATE  "STATE The current state of the system" %
%   N9:6  SYSTEM_PURGE %
%   N7:29  GETTER_HTI_ALM_DLY %
%   T4:56  GETTER_1_HTI_ALM_TMR %
%   B26:17/5  GET_1_HTI_ALARM %
%   B26:5/7  GETTER_HTI_WRN_EN %
%   N7:30  GETTER_HTI_WRN_DLY %
%   T4:57  GETTER_1_HTI_WRN_TMR %
%   B26:23/5  GET_1_HTI_WARN %
% Rung: 9 %
% TITLE: OPEN TC's %
SOR EQU I:4.7 N7:81 XIC B26:3/1 BST MOV N7:31 T4:128.PRE NXB TON T4:128 1.0 5 0 NXB XIC T4:128/DN OTE B26:20/0 BND EOR
%   I:4.7  GET_1_PH_INNER_TC  "TC1" %
%   N7:81  TC_OPEN_SP  "CONFIG The value read by an open TC input" %
%   B26:3/1  OPEN_TC1_ALARM_EN  "CONFIG open TC" %
%   N7:31  OPEN_TC_DLY %
%   T4:128  OPEN_TC1_TMR %
%   B26:20/0  OPEN_TC1_ALARM %

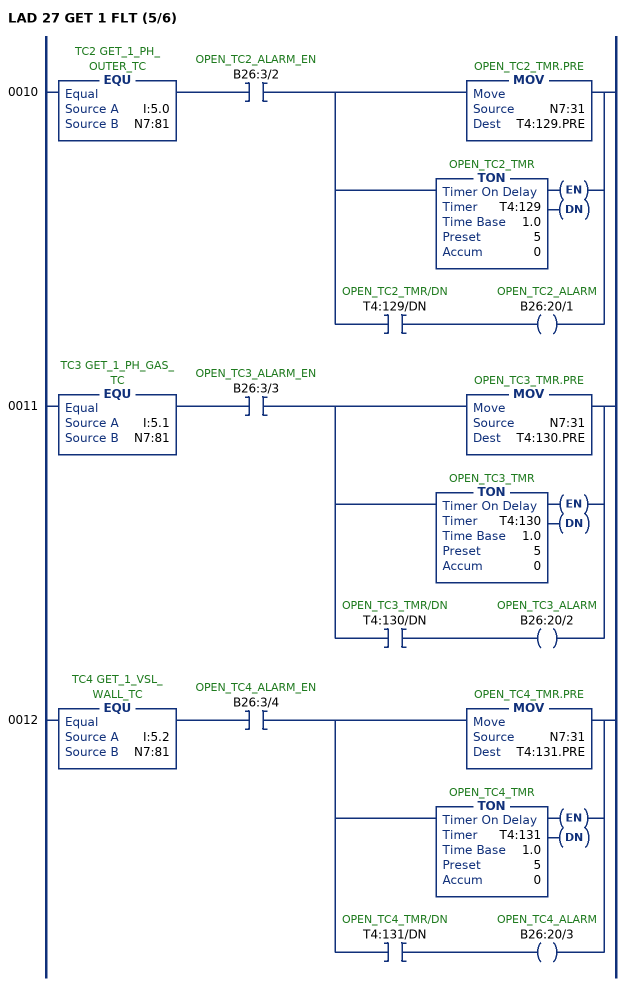
% Rung: 10 %
SOR EQU I:5.0 N7:81 XIC B26:3/2 BST MOV N7:31 T4:129.PRE NXB TON T4:129 1.0 5 0 NXB XIC T4:129/DN OTE B26:20/1 BND EOR
%   I:5.0  GET_1_PH_OUTER_TC  "TC2" %
%   N7:81  TC_OPEN_SP  "CONFIG The value read by an open TC input" %
%   B26:3/2  OPEN_TC2_ALARM_EN %
%   N7:31  OPEN_TC_DLY %
%   T4:129  OPEN_TC2_TMR %
%   B26:20/1  OPEN_TC2_ALARM %
% Rung: 11 %
SOR EQU I:5.1 N7:81 XIC B26:3/3 BST MOV N7:31 T4:130.PRE NXB TON T4:130 1.0 5 0 NXB XIC T4:130/DN OTE B26:20/2 BND EOR
%   I:5.1  GET_1_PH_GAS_TC  "TC3" %
%   N7:81  TC_OPEN_SP  "CONFIG The value read by an open TC input" %
%   B26:3/3  OPEN_TC3_ALARM_EN %
%   N7:31  OPEN_TC_DLY %
%   T4:130  OPEN_TC3_TMR %
%   B26:20/2  OPEN_TC3_ALARM %
% Rung: 12 %
SOR EQU I:5.2 N7:81 XIC B26:3/4 BST MOV N7:31 T4:131.PRE NXB TON T4:131 1.0 5 0 NXB XIC T4:131/DN OTE B26:20/3 BND EOR
%   I:5.2  GET_1_VSL_WALL_TC  "TC4" %
%   N7:81  TC_OPEN_SP  "CONFIG The value read by an open TC input" %
%   B26:3/4  OPEN_TC4_ALARM_EN %
%   N7:31  OPEN_TC_DLY %
%   T4:131  OPEN_TC4_TMR %
%   B26:20/3  OPEN_TC4_ALARM %

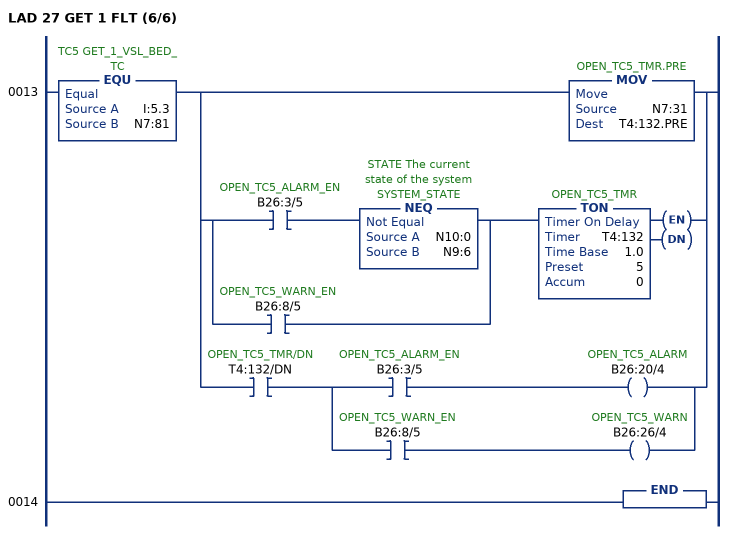
% Rung: 13 %
SOR EQU I:5.3 N7:81 BST MOV N7:31 T4:132.PRE NXB BST XIC B26:3/5 NEQ N10:0 N9:6 NXB XIC B26:8/5 BND TON T4:132 1.0 5 0 NXB XIC T4:132/DN BST XIC B26:3/5 OTE B26:20/4 NXB XIC B26:8/5 OTE B26:26/4 BND BND EOR
%   I:5.3  GET_1_VSL_BED_TC  "TC5" %
%   N7:81  TC_OPEN_SP  "CONFIG The value read by an open TC input" %
%   N7:31  OPEN_TC_DLY %
%   T4:132  OPEN_TC5_TMR %
%   B26:3/5  OPEN_TC5_ALARM_EN %
%   N10:0  SYSTEM_STATE  "STATE The current state of the system" %
%   N9:6  SYSTEM_PURGE %
%   B26:8/5  OPEN_TC5_WARN_EN %
%   B26:20/4  OPEN_TC5_ALARM %
%   B26:26/4  OPEN_TC5_WARN %
% Rung: 14 %
SOR END EOR

LADDER 28 "GET 1"
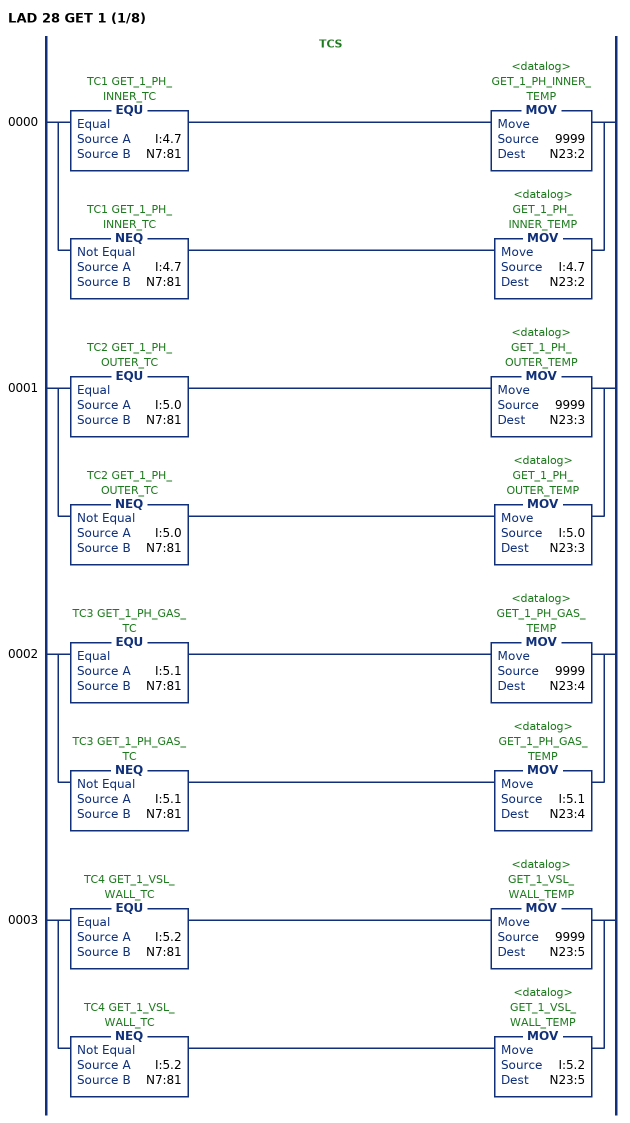
% Rung: 0 %
% TITLE: TCS %
SOR BST EQU I:4.7 N7:81 MOV 9999 N23:2 NXB NEQ I:4.7 N7:81 MOV I:4.7 N23:2 BND EOR
%   I:4.7  GET_1_PH_INNER_TC  "TC1" %
%   N7:81  TC_OPEN_SP  "CONFIG The value read by an open TC input" %
%   N23:2  GET_1_PH_INNER_TEMP  "<datalog>" %
% Rung: 1 %
SOR BST EQU I:5.0 N7:81 MOV 9999 N23:3 NXB NEQ I:5.0 N7:81 MOV I:5.0 N23:3 BND EOR
%   I:5.0  GET_1_PH_OUTER_TC  "TC2" %
%   N7:81  TC_OPEN_SP  "CONFIG The value read by an open TC input" %
%   N23:3  GET_1_PH_OUTER_TEMP  "<datalog>" %
% Rung: 2 %
SOR BST EQU I:5.1 N7:81 MOV 9999 N23:4 NXB NEQ I:5.1 N7:81 MOV I:5.1 N23:4 BND EOR
%   I:5.1  GET_1_PH_GAS_TC  "TC3" %
%   N7:81  TC_OPEN_SP  "CONFIG The value read by an open TC input" %
%   N23:4  GET_1_PH_GAS_TEMP  "<datalog>" %
% Rung: 3 %
SOR BST EQU I:5.2 N7:81 MOV 9999 N23:5 NXB NEQ I:5.2 N7:81 MOV I:5.2 N23:5 BND EOR
%   I:5.2  GET_1_VSL_WALL_TC  "TC4" %
%   N7:81  TC_OPEN_SP  "CONFIG The value read by an open TC input" %
%   N23:5  GET_1_VSL_WALL_TEMP  "<datalog>" %

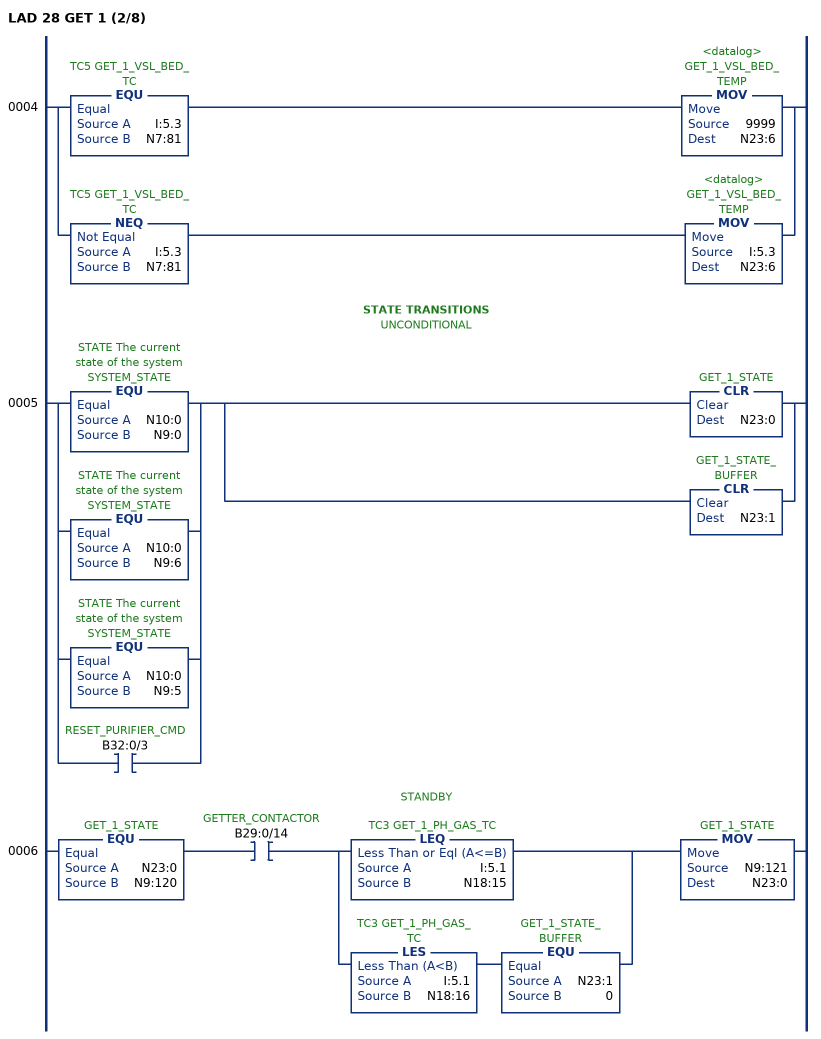
% Rung: 4 %
SOR BST EQU I:5.3 N7:81 MOV 9999 N23:6 NXB NEQ I:5.3 N7:81 MOV I:5.3 N23:6 BND EOR
%   I:5.3  GET_1_VSL_BED_TC  "TC5" %
%   N7:81  TC_OPEN_SP  "CONFIG The value read by an open TC input" %
%   N23:6  GET_1_VSL_BED_TEMP  "<datalog>" %
% Rung: 5 %
% TITLE: STATE TRANSITIONS %
% UNCONDITIONAL %
SOR BST EQU N10:0 N9:0 NXB EQU N10:0 N9:6 NXB EQU N10:0 N9:5 NXB XIC B32:0/3 BND BST CLR N23:0 NXB CLR N23:1 BND EOR
%   N10:0  SYSTEM_STATE  "STATE The current state of the system" %
%   N9:0  SYSTEM_OFFLINE %
%   N9:6  SYSTEM_PURGE %
%   N9:5  SYSTEM_QUICK_START %
%   B32:0/3  RESET_PURIFIER_CMD %
%   N23:0  GET_1_STATE %
%   N23:1  GET_1_STATE_BUFFER %
% Rung: 6 %
% STANDBY %
SOR EQU N23:0 N9:120 XIC B29:0/14 BST LEQ I:5.1 N18:15 NXB LES I:5.1 N18:16 EQU N23:1 0 BND MOV N9:121 N23:0 EOR
%   N23:0  GET_1_STATE %
%   N9:120  GETTER_STANDBY %
%   B29:0/14  GETTER_CONTACTOR %
%   I:5.1  GET_1_PH_GAS_TC  "TC3" %
%   N18:15  GETTER_SS_BEGIN_TEMP %
%   N18:16  GETTER_SS_END_TEMP %
%   N23:1  GET_1_STATE_BUFFER %
%   N9:121  GETTER_SOFTSTART %

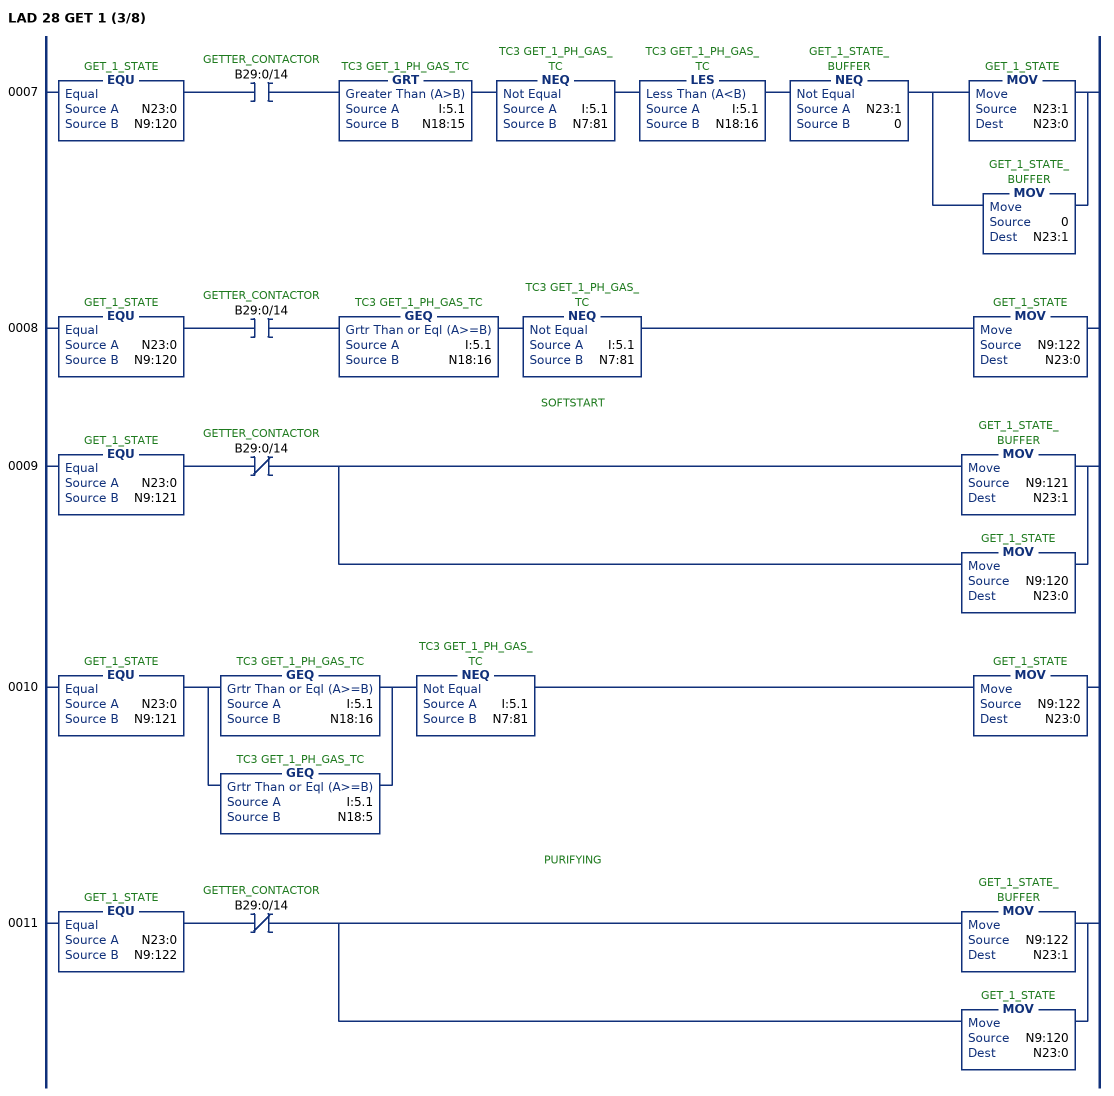
% Rung: 7 %
SOR EQU N23:0 N9:120 XIC B29:0/14 GRT I:5.1 N18:15 NEQ I:5.1 N7:81 LES I:5.1 N18:16 NEQ N23:1 0 BST MOV N23:1 N23:0 NXB MOV 0 N23:1 BND EOR
%   N23:0  GET_1_STATE %
%   N9:120  GETTER_STANDBY %
%   B29:0/14  GETTER_CONTACTOR %
%   I:5.1  GET_1_PH_GAS_TC  "TC3" %
%   N18:15  GETTER_SS_BEGIN_TEMP %
%   N7:81  TC_OPEN_SP  "CONFIG The value read by an open TC input" %
%   N18:16  GETTER_SS_END_TEMP %
%   N23:1  GET_1_STATE_BUFFER %
% Rung: 8 %
SOR EQU N23:0 N9:120 XIC B29:0/14 GEQ I:5.1 N18:16 NEQ I:5.1 N7:81 MOV N9:122 N23:0 EOR
%   N23:0  GET_1_STATE %
%   N9:120  GETTER_STANDBY %
%   B29:0/14  GETTER_CONTACTOR %
%   I:5.1  GET_1_PH_GAS_TC  "TC3" %
%   N18:16  GETTER_SS_END_TEMP %
%   N7:81  TC_OPEN_SP  "CONFIG The value read by an open TC input" %
%   N9:122  GETTER_PURIFYING %
% Rung: 9 %
% SOFTSTART %
SOR EQU N23:0 N9:121 XIO B29:0/14 BST MOV N9:121 N23:1 NXB MOV N9:120 N23:0 BND EOR
%   N23:0  GET_1_STATE %
%   N9:121  GETTER_SOFTSTART %
%   B29:0/14  GETTER_CONTACTOR %
%   N23:1  GET_1_STATE_BUFFER %
%   N9:120  GETTER_STANDBY %
% Rung: 10 %
SOR EQU N23:0 N9:121 BST GEQ I:5.1 N18:16 NXB GEQ I:5.1 N18:5 BND NEQ I:5.1 N7:81 MOV N9:122 N23:0 EOR
%   N23:0  GET_1_STATE %
%   N9:121  GETTER_SOFTSTART %
%   I:5.1  GET_1_PH_GAS_TC  "TC3" %
%   N18:16  GETTER_SS_END_TEMP %
%   N18:5  GETTER_PH_SP  "<datalog>" %
%   N7:81  TC_OPEN_SP  "CONFIG The value read by an open TC input" %
%   N9:122  GETTER_PURIFYING %
% Rung: 11 %
% PURIFYING %
SOR EQU N23:0 N9:122 XIO B29:0/14 BST MOV N9:122 N23:1 NXB MOV N9:120 N23:0 BND EOR
%   N23:0  GET_1_STATE %
%   N9:122  GETTER_PURIFYING %
%   B29:0/14  GETTER_CONTACTOR %
%   N23:1  GET_1_STATE_BUFFER %
%   N9:120  GETTER_STANDBY %

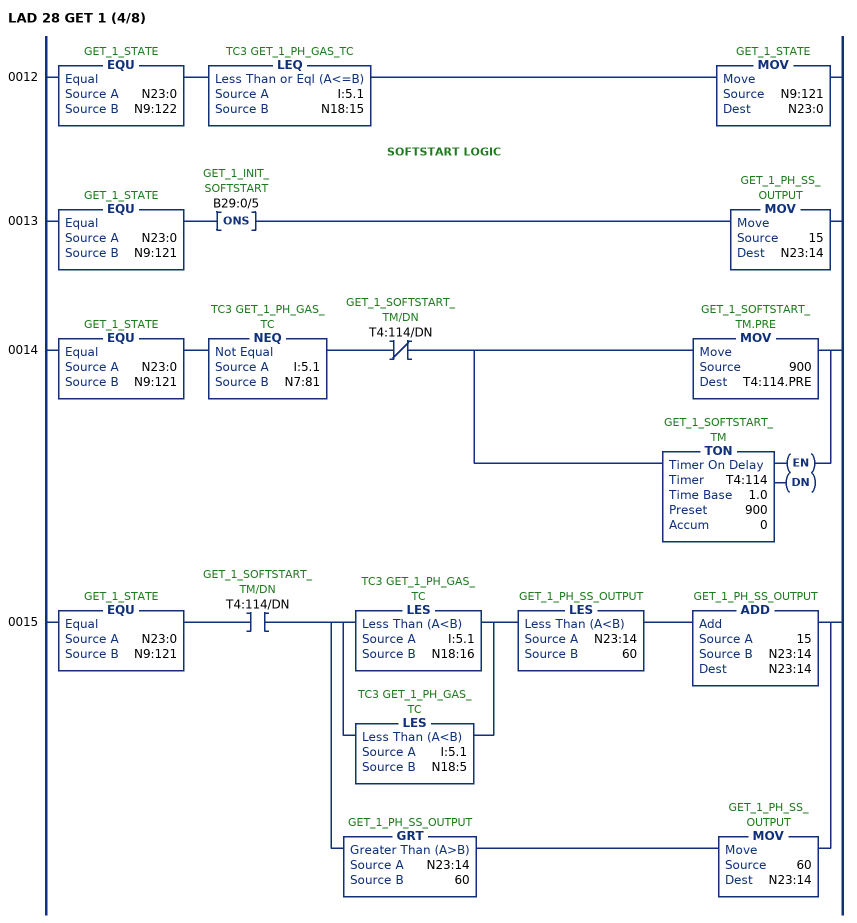
% Rung: 12 %
SOR EQU N23:0 N9:122 LEQ I:5.1 N18:15 MOV N9:121 N23:0 EOR
%   N23:0  GET_1_STATE %
%   N9:122  GETTER_PURIFYING %
%   I:5.1  GET_1_PH_GAS_TC  "TC3" %
%   N18:15  GETTER_SS_BEGIN_TEMP %
%   N9:121  GETTER_SOFTSTART %
% Rung: 13 %
% TITLE: SOFTSTART LOGIC %
SOR EQU N23:0 N9:121 ONS B29:0/5 MOV 15 N23:14 EOR
%   N23:0  GET_1_STATE %
%   N9:121  GETTER_SOFTSTART %
%   B29:0/5  GET_1_INIT_SOFTSTART %
%   N23:14  GET_1_PH_SS_OUTPUT %
% Rung: 14 %
SOR EQU N23:0 N9:121 NEQ I:5.1 N7:81 XIO T4:114/DN BST MOV 900 T4:114.PRE NXB TON T4:114 1.0 900 0 BND EOR
%   N23:0  GET_1_STATE %
%   N9:121  GETTER_SOFTSTART %
%   I:5.1  GET_1_PH_GAS_TC  "TC3" %
%   N7:81  TC_OPEN_SP  "CONFIG The value read by an open TC input" %
%   T4:114  GET_1_SOFTSTART_TM %
% Rung: 15 %
SOR EQU N23:0 N9:121 XIC T4:114/DN BST BST LES I:5.1 N18:16 NXB LES I:5.1 N18:5 BND LES N23:14 60 ADD 15 N23:14 N23:14 NXB GRT N23:14 60 MOV 60 N23:14 BND EOR
%   N23:0  GET_1_STATE %
%   N9:121  GETTER_SOFTSTART %
%   T4:114  GET_1_SOFTSTART_TM %
%   I:5.1  GET_1_PH_GAS_TC  "TC3" %
%   N18:16  GETTER_SS_END_TEMP %
%   N18:5  GETTER_PH_SP  "<datalog>" %
%   N23:14  GET_1_PH_SS_OUTPUT %

